(* IEC 61131-3 sources: Industry-PLC-LLM/data/PLCBEAD_repo/PLCBEAD_PLCEmbed-main/PLC-BEAD/Source/GEB/Network_IP4_CHECK, 1 file *)

(* ---- IP4_CHECK.ST ---- *)
FUNCTION IP4_CHECK:BOOL

	VAR_INPUT
		NIP :	DWORD;
		LIP :	DWORD;
		SM :	DWORD;
	END_VAR

	IP4_CHECK := (NIP AND sm) = (LIP AND SM);

END_FUNCTION

PROGRAM program0
	VAR
		NIP :	DWORD;
		LIP :	DWORD;
		SM :	DWORD;
		CEIL5_OUT : BOOL;
	END_VAR

  	CEIL5_OUT := IP4_CHECK(NIP, LIP, SM);
END_PROGRAM
